PROGRAM WeatherStation
VAR
	fbThiesWSC11					:FB_ThiesWSC11;
	fbThiesWSC11Time				:FB_ThiesWSC11Time;
	fbEB_Time						:FB_EB_Time;
	fbThresholdSwitch				:ARRAY[1..8] OF FB_ThresholdSwitch;
	fbWeeklyTimeSwitch				:ARRAY[1..2] OF FB_WeeklyTimeSwitch;
	bResetWSC11						:BOOL;
	bSetTimeManual					:BOOL;

	//FBs für Aktion A_Sonnenposition
	fbCalcSunPosition				:FB_CalcSunPosition;
	fbThresholdswitch_Beschattung	:ARRAY[1..4] OF FB_Thresholdswitch;
	R_TRIG							:ARRAY[1..4] OF R_TRIG;;
	TOF								:ARRAY[1..4] OF TOF;
	bTest_West						:BOOL := FALSE;
	bTest_Sued						:BOOL := FALSE;
	bTest_Osten						:BOOL := FALSE;
	bTestSafetyPosition				:BOOL := FALSE;
	bTestSafetyPositionMarkise		:BOOL := FALSE;
	bTest: BOOL;
END_VAR

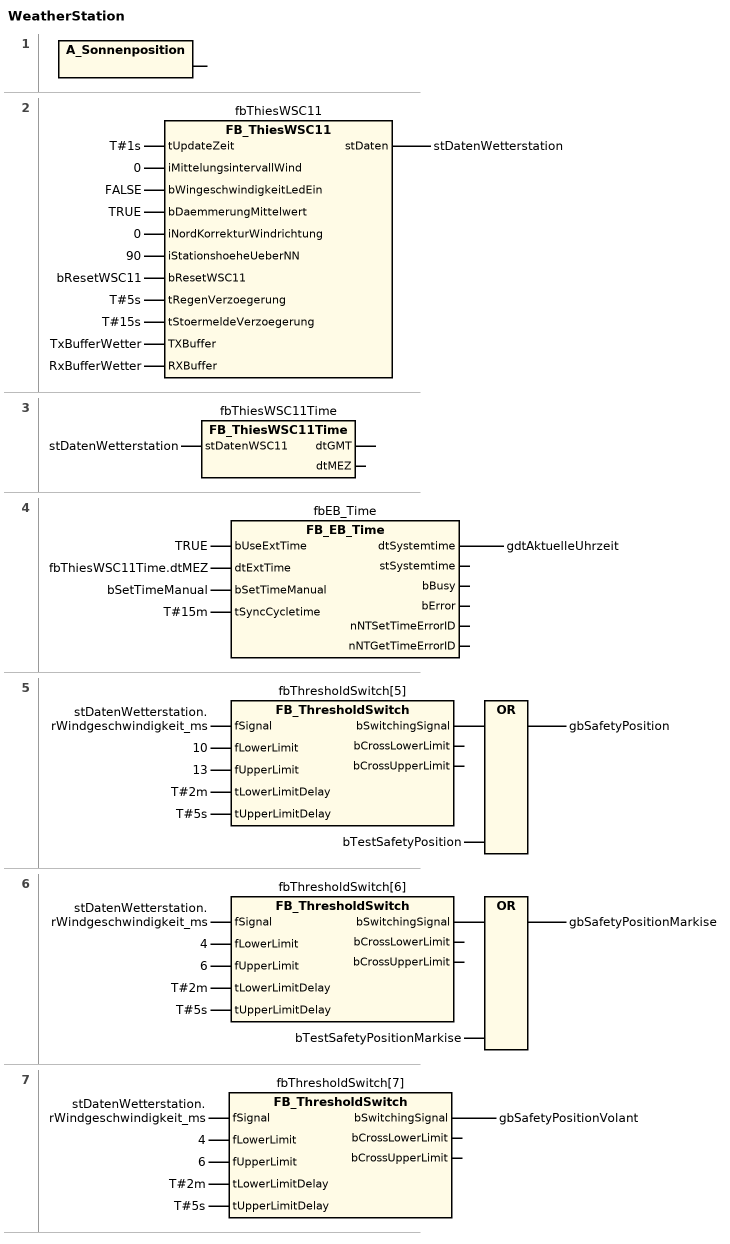
// NETWORK 1
A_Sonnenposition();

// NETWORK 2
fbThiesWSC11(
    tUpdateZeit := T#1s,
    iMittelungsintervallWind := 0,
    bWingeschwindigkeitLedEin := FALSE,
    bDaemmerungMittelwert := TRUE,
    iNordKorrekturWindrichtung := 0,
    iStationshoeheUeberNN := 90,
    bResetWSC11 := bResetWSC11,
    tRegenVerzoegerung := T#5s,
    tStoermeldeVerzoegerung := T#15s,
    TXBuffer := TxBufferWetter,
    RXBuffer := RxBufferWetter); // FB_ThiesWSC11
stDatenWetterstation := fbThiesWSC11.stDaten;

// NETWORK 3
fbThiesWSC11Time(stDatenWSC11 := stDatenWetterstation); // FB_ThiesWSC11Time

// NETWORK 4
fbEB_Time(
    bUseExtTime := TRUE,
    dtExtTime := fbThiesWSC11Time.dtMEZ,
    bSetTimeManual := bSetTimeManual,
    tSyncCycletime := T#15m); // FB_EB_Time
gdtAktuelleUhrzeit := fbEB_Time.dtSystemtime;

// NETWORK 5
fbThresholdSwitch[5](
    fSignal := stDatenWetterstation.rWindgeschwindigkeit_ms,
    fLowerLimit := 10,
    fUpperLimit := 13,
    tLowerLimitDelay := T#2m,
    tUpperLimitDelay := T#5s); // FB_ThresholdSwitch
gbSafetyPosition := fbThresholdSwitch[5].bSwitchingSignal OR bTestSafetyPosition;

// NETWORK 6
fbThresholdSwitch[6](
    fSignal := stDatenWetterstation.rWindgeschwindigkeit_ms,
    fLowerLimit := 4,
    fUpperLimit := 6,
    tLowerLimitDelay := T#2m,
    tUpperLimitDelay := T#5s); // FB_ThresholdSwitch
gbSafetyPositionMarkise := fbThresholdSwitch[6].bSwitchingSignal OR bTestSafetyPositionMarkise;

// NETWORK 7
fbThresholdSwitch[7](
    fSignal := stDatenWetterstation.rWindgeschwindigkeit_ms,
    fLowerLimit := 4,
    fUpperLimit := 6,
    tLowerLimitDelay := T#2m,
    tUpperLimitDelay := T#5s); // FB_ThresholdSwitch
gbSafetyPositionVolant := fbThresholdSwitch[7].bSwitchingSignal;

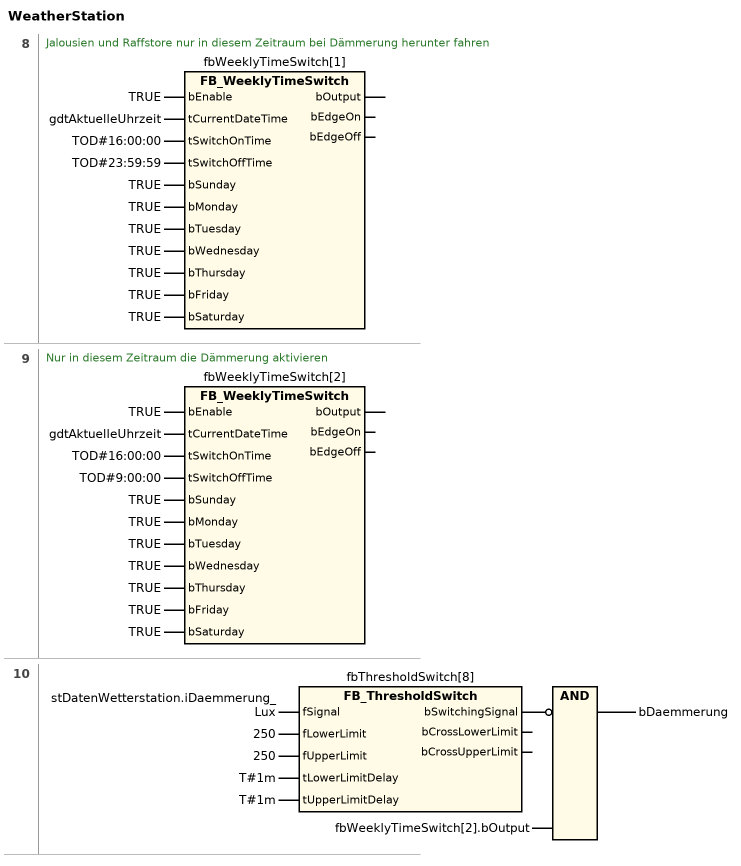
// NETWORK 8
// Jalousien und Raffstore nur in diesem Zeitraum bei Dämmerung herunter fahren
fbWeeklyTimeSwitch[1](
    bEnable := TRUE,
    tCurrentDateTime := gdtAktuelleUhrzeit,
    tSwitchOnTime := TOD#16:00:00,
    tSwitchOffTime := TOD#23:59:59,
    bSunday := TRUE,
    bMonday := TRUE,
    bTuesday := TRUE,
    bWednesday := TRUE,
    bThursday := TRUE,
    bFriday := TRUE,
    bSaturday := TRUE); // FB_WeeklyTimeSwitch

// NETWORK 9
// Nur in diesem Zeitraum die Dämmerung aktivieren
fbWeeklyTimeSwitch[2](
    bEnable := TRUE,
    tCurrentDateTime := gdtAktuelleUhrzeit,
    tSwitchOnTime := TOD#16:00:00,
    tSwitchOffTime := TOD#9:00:00,
    bSunday := TRUE,
    bMonday := TRUE,
    bTuesday := TRUE,
    bWednesday := TRUE,
    bThursday := TRUE,
    bFriday := TRUE,
    bSaturday := TRUE); // FB_WeeklyTimeSwitch

// NETWORK 10
fbThresholdSwitch[8](
    fSignal := stDatenWetterstation.iDaemmerung_Lux,
    fLowerLimit := 250,
    fUpperLimit := 250,
    tLowerLimitDelay := T#1m,
    tUpperLimitDelay := T#1m); // FB_ThresholdSwitch
bDaemmerung := NOT fbThresholdSwitch[8].bSwitchingSignal AND fbWeeklyTimeSwitch[2].bOutput;

ACTION A_Sonnenposition:
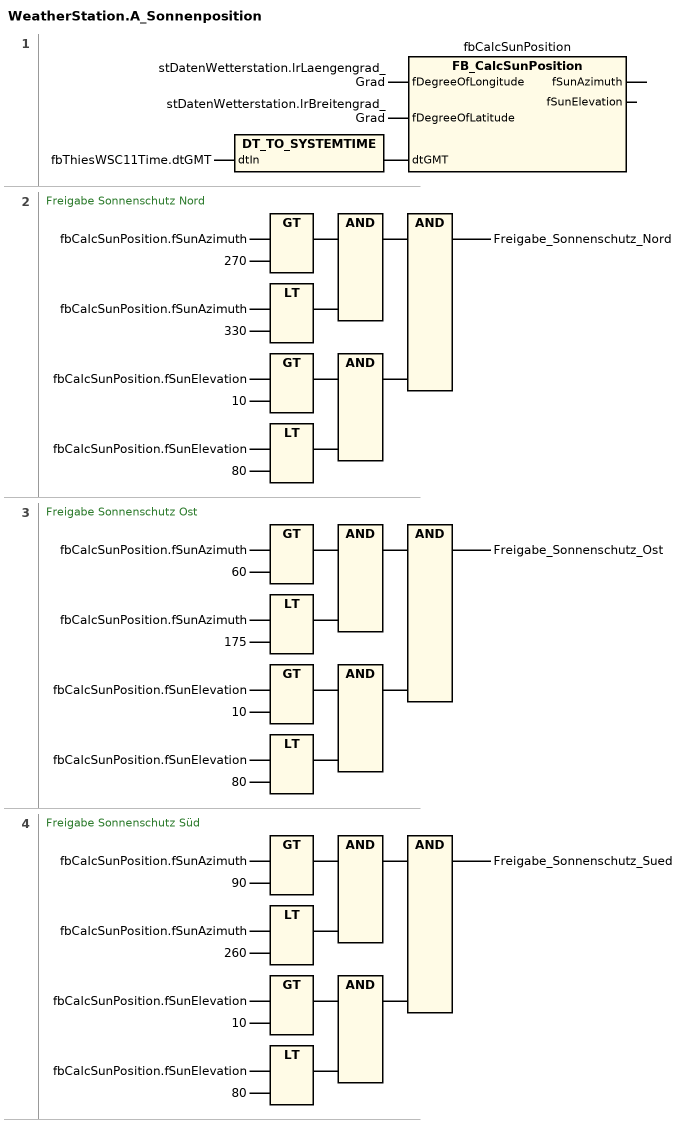
// NETWORK 1
fbCalcSunPosition(
    fDegreeOfLongitude := stDatenWetterstation.lrLaengengrad_Grad,
    fDegreeOfLatitude := stDatenWetterstation.lrBreitengrad_Grad,
    dtGMT := DT_TO_SYSTEMTIME(dtIn := fbThiesWSC11Time.dtGMT)); // FB_CalcSunPosition

// NETWORK 2
// Freigabe Sonnenschutz Nord
Freigabe_Sonnenschutz_Nord := (fbCalcSunPosition.fSunAzimuth > 270 AND fbCalcSunPosition.fSunAzimuth < 330) AND (fbCalcSunPosition.fSunElevation > 10 AND fbCalcSunPosition.fSunElevation < 80);

// NETWORK 3
// Freigabe Sonnenschutz Ost
Freigabe_Sonnenschutz_Ost := (fbCalcSunPosition.fSunAzimuth > 60 AND fbCalcSunPosition.fSunAzimuth < 175) AND (fbCalcSunPosition.fSunElevation > 10 AND fbCalcSunPosition.fSunElevation < 80);

// NETWORK 4
// Freigabe Sonnenschutz Süd
Freigabe_Sonnenschutz_Sued := (fbCalcSunPosition.fSunAzimuth > 90 AND fbCalcSunPosition.fSunAzimuth < 260) AND (fbCalcSunPosition.fSunElevation > 10 AND fbCalcSunPosition.fSunElevation < 80);

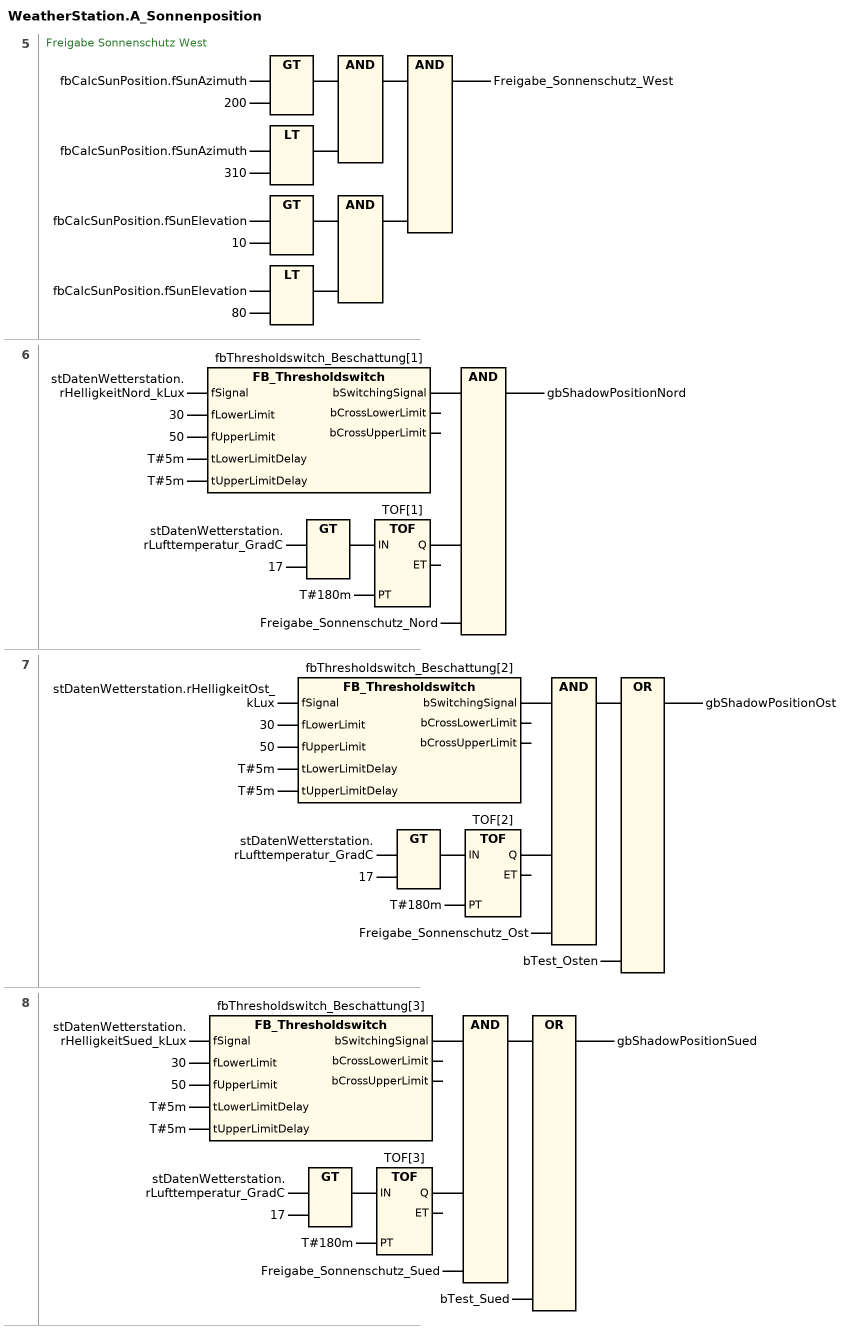
// NETWORK 5
// Freigabe Sonnenschutz West
Freigabe_Sonnenschutz_West := (fbCalcSunPosition.fSunAzimuth > 200 AND fbCalcSunPosition.fSunAzimuth < 310) AND (fbCalcSunPosition.fSunElevation > 10 AND fbCalcSunPosition.fSunElevation < 80);

// NETWORK 6
fbThresholdswitch_Beschattung[1](
    fSignal := stDatenWetterstation.rHelligkeitNord_kLux,
    fLowerLimit := 30,
    fUpperLimit := 50,
    tLowerLimitDelay := T#5m,
    tUpperLimitDelay := T#5m); // FB_Thresholdswitch
TOF[1](IN := stDatenWetterstation.rLufttemperatur_GradC > 17, PT := T#180m); // TOF
gbShadowPositionNord := fbThresholdswitch_Beschattung[1].bSwitchingSignal AND TOF[1].Q AND Freigabe_Sonnenschutz_Nord;

// NETWORK 7
fbThresholdswitch_Beschattung[2](
    fSignal := stDatenWetterstation.rHelligkeitOst_kLux,
    fLowerLimit := 30,
    fUpperLimit := 50,
    tLowerLimitDelay := T#5m,
    tUpperLimitDelay := T#5m); // FB_Thresholdswitch
TOF[2](IN := stDatenWetterstation.rLufttemperatur_GradC > 17, PT := T#180m); // TOF
gbShadowPositionOst := fbThresholdswitch_Beschattung[2].bSwitchingSignal AND TOF[2].Q AND Freigabe_Sonnenschutz_Ost OR bTest_Osten;

// NETWORK 8
fbThresholdswitch_Beschattung[3](
    fSignal := stDatenWetterstation.rHelligkeitSued_kLux,
    fLowerLimit := 30,
    fUpperLimit := 50,
    tLowerLimitDelay := T#5m,
    tUpperLimitDelay := T#5m); // FB_Thresholdswitch
TOF[3](IN := stDatenWetterstation.rLufttemperatur_GradC > 17, PT := T#180m); // TOF
gbShadowPositionSued := fbThresholdswitch_Beschattung[3].bSwitchingSignal AND TOF[3].Q AND Freigabe_Sonnenschutz_Sued OR bTest_Sued;

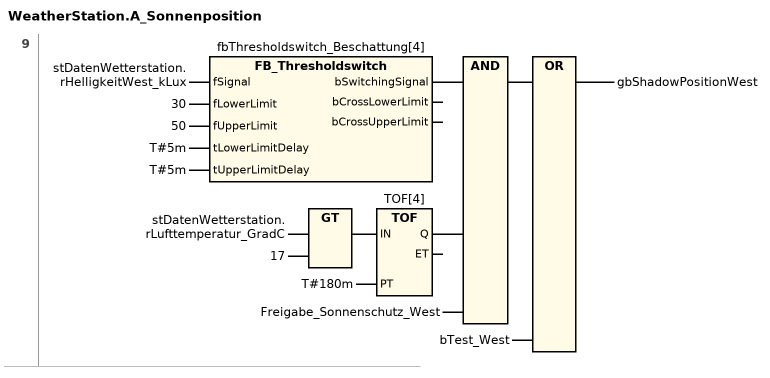
// NETWORK 9
fbThresholdswitch_Beschattung[4](
    fSignal := stDatenWetterstation.rHelligkeitWest_kLux,
    fLowerLimit := 30,
    fUpperLimit := 50,
    tLowerLimitDelay := T#5m,
    tUpperLimitDelay := T#5m); // FB_Thresholdswitch
TOF[4](IN := stDatenWetterstation.rLufttemperatur_GradC > 17, PT := T#180m); // TOF
gbShadowPositionWest := fbThresholdswitch_Beschattung[4].bSwitchingSignal AND TOF[4].Q AND Freigabe_Sonnenschutz_West OR bTest_West;
END_ACTION

END_PROGRAM

(* stored: Version 1.1.0.1, ProductVersion 3.1.4024.12
   POU WeatherStation: Id {25647cf7-b494-44c8-b6a5-90c59c6e154e}, SpecialFunc None
   Action A_Sonnenposition: Id {d069584f-bce7-427d-bc1a-9570778e8af5} *)
